TYPE udt_Generic_Nok_Data_Grid_20251208 :
STRUCT
	TimeStamp : STRING;
	Model_ID : STRING;
	NOK_Faulted : STRING;    
	Unload_Completed : BOOL; (*reset signal*)
	
END_STRUCT
END_TYPE

(* stored: Version 1.1.0.1, ProductVersion 3.1.4024.12
   DUT udt_Generic_Nok_Data_Grid_20251208: Id {56ebabc9-fa02-454e-8e18-8d08bcec7a17} *)
